// TIA Portal V17 export
// export: Created 2022-07-20T07:02:36.4789637Z, ExportSetting WithDefaults, DisplayName Totally Integrated Automation Portal, DisplayVersion V17, DisplayName TIA Portal Openness, DisplayVersion V17, DisplayName TIA Portal Version Control Interface, DisplayVersion V17, DisplayName SINAMICS Startdrive Advanced, DisplayVersion V17, DisplayName SINAMICS Startdrive G130, G150, S120, S150, SINAMICS MV, S210, DisplayVersion V17, DisplayName SINAMICS Startdrive G110M, G120, G120C, G120D, G120P, G115D, DisplayVersion V17, DisplayName STEP 7 Professional, DisplayVersion V17, DisplayName STEP 7 Safety, DisplayVersion V17, DisplayName WinCC Advanced, DisplayVersion V17
VAR_GLOBAL   // PLC tag table "IFM_DV2510"
END_VAR
VAR_GLOBAL CONSTANT   // user constants
   SEGMENT_LED_OFF : Byte := 0;
   SEGMENT_LED_BLUE : Byte := 1;
   SEGMENT_LED_GREEN : Byte := 2;
   SEGMENT_LED_TURQUOISE : Byte := 3;
   SEGMENT_LED_RED : Byte := 4;
   SEGMENT_LED_VIOLET : Byte := 5;
   SEGMENT_LED_ORANGE : Byte := 6;
   SEGMENT_LED_WHITE : Byte := 7;
   SEGMENT_LED_YELLOW : Byte := 8;
   SEGMENT_LED_PERMANENT_ON : Byte := 0;
   SEGMENT_LED_SLOW_BLINKING : Byte := 16;
   SEGMENT_LED_NORMAL_BLINKING : Byte := 32;
   SEGMENT_LED_QUICK_BLINKING : Byte := 48;
   SEGMENT_LED_SLOW_FLASH : Byte := 64;
   SEGMENT_LED_NORMAL_FLASH : Byte := 80;
   SEGMENT_LED_QUICK_FLASH : Byte := 96;
END_VAR
